// TwinCAT 3 PLC project PRG_B_IODecorator
// Title: B_IODecorator
// Company: RafalOS
// Author: Rafał Osajda
// ProjectVersion: 0.0.0.3
// ProgramVersion: 3.1.4024.0
// libraries:
//   B_Base, * (RafalOS)
//   B_BaseDecorate, * (RafalOS)
//   B_IO, * (RafalOS)
//   Tc2_Standard, * (Beckhoff Automation GmbH)
//   Tc2_System, * (Beckhoff Automation GmbH)
//   Tc3_Module, * (Beckhoff Automation GmbH)
// project tree:
//   / PlcTask.TcTTO (not stored)
//   POUs Compilation/ PRG_Compilation.TcPOU
//   POUs/Sensor/ FB_Sensor_TestParentDecorator.TcPOU, FB_Sensor_NO_TestDecorator.TcPOU (not stored), FB_Sensor_NC_TestDecorator.TcPOU, FB_Sensor_NO_2InRow_TestDecorator.TcPOU, ITF_Sensor_TestDecorator.TcIO, ITF_Sensor_NO_2InRow_TestDecorator.TcIO (not stored)

// ---- POUs/Sensor/ITF_Sensor_TestDecorator.TcIO
INTERFACE ITF_Sensor_TestDecorator EXTENDS ITF_Sensor

METHOD PUBLIC SetContact
VAR_INPUT
	bIN: BOOL;
END_VAR
END_METHOD

END_INTERFACE

// ---- POUs Compilation/PRG_Compilation.TcPOU
PROGRAM PRG_Compilation
VAR
	senNO				: FB_Sensor_NO;
	senNO_DecoratorTest	: FB_Sensor_NO_TestDecorator (fbToDecorate := senNO);
	senNC				: FB_Sensor_NC;
	senNC_DecoratorTest	: FB_Sensor_NC_TestDecorator (fbToDecorate := senNC);
	sen2NO				: FB_Sensor_NO_2InRow;
	sen2NO_DecoratorTest: FB_Sensor_NO_2InRow_TestDecorator (fbToDecorate := sen2NO);
	
END_VAR

END_PROGRAM

// ---- POUs/Sensor/FB_Sensor_NC_TestDecorator.TcPOU
FUNCTION_BLOCK FB_Sensor_NC_TestDecorator EXTENDS FB_Sensor_TestParentDecorator 
VAR
	
END_VAR

(*			
	EVERDE sp. z o.o.
	Rafał Osajda		05.02.2025		TC 4026.13		wer. 0.0.0.1
	Zwraca aktualny stan czujnika
*)
METHOD IsActive : BOOL
IsActive			:= NOT THIS^.bContactTest;
END_METHOD

END_FUNCTION_BLOCK

// ---- POUs/Sensor/FB_Sensor_TestParentDecorator.TcPOU
FUNCTION_BLOCK ABSTRACT FB_Sensor_TestParentDecorator EXTENDS FB_BaseComponentDecoratorParent IMPLEMENTS ITF_Sensor_TestDecorator
VAR
	bContactTest			: BOOL;
END_VAR

(*			
	EVERDE sp. z o.o.
	Rafał Osajda		05.02.2025		TC 4026.13		wer. 0.0.0.1
	Zwraca aktualny stan czujnika
*)
METHOD IsActive : BOOL
END_METHOD

METHOD PUBLIC SetContact
VAR_INPUT
	bIN: BOOL;
END_VAR
THIS^.bContactTest		:= bIN;
END_METHOD

END_FUNCTION_BLOCK

// ---- POUs/Sensor/FB_Sensor_NO_2InRow_TestDecorator.TcPOU
FUNCTION_BLOCK FB_Sensor_NO_2InRow_TestDecorator EXTENDS FB_Sensor_TestParentDecorator IMPLEMENTS ITF_Sensor_NO_2InRow_TestDecorator
VAR
	bContact2Test			: BOOL;
END_VAR

(*			
	EVERDE sp. z o.o.
	Rafał Osajda		05.02.2025		TC 4026.13		wer. 0.0.0.1
	Zwraca aktualny stan czujnika
*)
METHOD IsActive : BOOL
IsActive			:= THIS^.bContactTest AND THIS^.bContact2Test;
END_METHOD

METHOD PUBLIC SetContact2
VAR_INPUT
	bIN: BOOL;
END_VAR
THIS^.bContact2Test		:= bIN;
END_METHOD

END_FUNCTION_BLOCK
